TYPE Room_Ctx_Io_Out :
STRUCT
	bPump			: BOOL;
	bBurner			: BOOL;
END_STRUCT
END_TYPE

(* stored: Version 1.1.0.1
   DUT Room_Ctx_Io_Out: Id {1da64ebc-f5ae-4ace-8e69-a586f42746cc} *)
